// TIA Portal V20 export
DATA_BLOCK "F-DB_DigitalOutput"   // DB111, F_DB
// stored: AutoNumber false, InstanceOfName F-FB_DigitalOutput, InstanceOfType FB
"F-FB_DigitalOutput"
BEGIN
END_DATA_BLOCK
